PROGRAM MAIN
VAR
END_VAR

BLOCK_CALL();

END_PROGRAM

(* stored: Version 1.1.0.1, ProductVersion 3.1.4024.16
   POU MAIN: Id {92c9fc8f-4654-4ad0-948d-9ff3b457c2f5}, SpecialFunc None *)
